INTERFACE I_OutputPort EXTENDS I_Disposable, I_EventEmitter, I_Serializable, I_HostMetadata

METHOD PUBLIC Accept
VAR_INPUT
	Visitor : I_OutputPortVisitor;
END_VAR
END_METHOD

PROPERTY PUBLIC Data : I_Datatype
GET
END_GET
END_PROPERTY

PROPERTY PUBLIC Name : T_MAXSTRING
GET
END_GET
END_PROPERTY

END_INTERFACE

(* stored: Version 1.1.0.1, ProductVersion 3.1.4024.12
   Itf I_OutputPort: Id {54edf811-4913-4b57-ba71-6036e501fb67}
   Method Accept: Id {aa3a9d71-ac12-40dd-ad8f-9235d7b1a13a}
   Property Data: Id {34ffee89-5c75-49b2-aafa-017e8e6186a1}
   Get Get: Id {10893aa1-b180-457a-9faf-31a7b60cc29a}
   Property Name: Id {8cad4439-74ed-46aa-b235-a0ecf44a87f8}
   Get Get: Id {a6c91baa-e710-4c9a-97ce-8dfb6515fb62} *)
